FUNCTION_BLOCK FB_Alarm
VAR_INPUT
	Alarm_Event: TcEventEntry;
	bInit : BOOL; 
    bRaise : BOOL; 
	bConfirm : BOOL; 
	bClear : BOOL; 
END_VAR
VAR
    fbAlarm : FB_TcAlarm; 
	sALarm : I_TcSourceInfo;
	bConfimed : BOOL;
END_VAR

IF bInit THEN
    bInit := FALSE; 
	bConfimed:= FALSE;
    fbAlarm.CreateEx(Alarm_Event, TRUE, sALarm); 
	fbAlarm.Confirm(0); 
END_IF

IF bRaise THEN 
    bRaise := FALSE; 
    fbAlarm.Raise(0); 
END_IF

IF bConfirm OR fbAlarm.eConfirmationState = 3 THEN
    bConfirm := FALSE; 
	bConfimed:= TRUE;
    fbAlarm.Confirm(0); 
END_IF

IF bClear THEN 
    bClear := FALSE; 
    fbAlarm.Clear(0, TRUE); 
END_IF

END_FUNCTION_BLOCK

(* stored: Version 1.1.0.1, ProductVersion 3.1.4024.9
   POU FB_Alarm: Id {8c391d5c-b5ef-4c7d-b904-008e97219267}, SpecialFunc None *)
